// TwinCAT 3 PLC project TcTransformTest
// ProgramVersion: 3.1.4023.0
// libraries:
//   Tc2_Standard, * (Beckhoff Automation GmbH)
//   Tc2_System, * (Beckhoff Automation GmbH)
//   Tc3_Module, * (Beckhoff Automation GmbH)
//   TcMatrix, * (Burks Engineering)
//   TcTransform, * (Burks Engineering)
//   TcUnit, * (www.tcunit.org)
// project tree:
//   / PlcTask.TcTTO
//   TESTs/ FB_Vector3_Test.TcPOU, FB_RMatrix_Test.TcPOU, FB_HMatrix_Test.TcPOU, PRG_TEST.TcPOU
// real-time tasks:
//   TASK PlcTask: cycle T#10ms, priority 20, ADS port 350

CONFIGURATION TcTransformTest
    RESOURCE PLC ON TwinCAT3
        TASK PlcTask(INTERVAL := T#10ms, PRIORITY := 20);
        PROGRAM PRG_TEST WITH PlcTask : PRG_TEST;
    END_RESOURCE
END_CONFIGURATION

// ---- TESTs/PRG_TEST.TcPOU
PROGRAM PRG_TEST
VAR
	fb_Vector3 : FB_Vector3_Test;
	fb_RMatrix : FB_RMatrix_Test;
	fb_HMatrix : FB_HMatrix_Test;
END_VAR

TcUnit.RUN();

END_PROGRAM

// ---- TESTs/FB_Vector3_Test.TcPOU
FUNCTION_BLOCK FB_Vector3_Test EXTENDS FB_TestSuite
VAR_INPUT
END_VAR
VAR_OUTPUT
END_VAR
VAR
END_VAR

WhenSetExpectValuesRetained();
WhenReversedExpectValuesReversed();
WhenCrossedExpectVectorOrthogonal();
WhenParallelCrossedExpectCleared();
WhenDottedExpectResult();

METHOD PRIVATE WhenCrossedExpectVectorOrthogonal
VAR_INPUT
END_VAR
VAR
	V1 : Vector3;
	V2 : Vector3;
	V3 : Vector3;
END_VAR
TEST('WhenCrossedExpectVectorOrthogonal');

// @TEST-RUN
V1.SetFromComponents(1,0,0);
V2.SetFromComponents(0,1,0);
V3 := V1.GetVector3CrossProduct(V2);

// @TEST-ASSERT
AssertTrue(V3.Z = 1,'cross product did not work');

TEST_FINISHED();
END_METHOD

METHOD PRIVATE WhenDottedExpectResult
VAR_INPUT
END_VAR
VAR
	V1 : Vector3;
	V2 : Vector3;
	V3 : Vector3;
	Dot : LREAL;
END_VAR
TEST('WhenDottedExpectResult');

// @TEST-RUN
V1.SetFromComponents(1,2,3);
V2 := V1;
Dot := V1.GetVector3DotProduct(V2);

// @TEST-ASSERT
AssertTrue(Dot = 14,'dot product did not work');

TEST_FINISHED();
END_METHOD

METHOD PRIVATE WhenParallelCrossedExpectCleared
VAR_INPUT
END_VAR
VAR
	V1 : Vector3;
	V2 : Vector3;
	V3 : Vector3;
END_VAR
TEST('WhenParallelCrossedExpectCleared');

// @TEST-RUN
V1.SetFromComponents(1,0,0);
V2.SetFromComponents(1,0,0);
V3 := V1.GetVector3CrossProduct(V2);

// @TEST-ASSERT
AssertTrue(V3.IsCleared,'parallel cross product is not zero');

TEST_FINISHED();
END_METHOD

METHOD PRIVATE WhenReversedExpectValuesReversed
VAR_INPUT
END_VAR
VAR
	V1 : Vector3;
	V2 : Vector3;
	V3 : Vector3;
END_VAR
TEST('WhenReversedExpectValuesReversed');

// @TEST-RUN
V1.SetFromComponents(1,2,3);
V2 := V1;
V1 := V1.GetReversed();//tests getter and reverse function
V3 := V2.GetVector3Sum(V2);

// @TEST-ASSERT
AssertTrue(V2.X + V1.X = 0,'Reversal did not work');
AssertTrue(V3.X = 2,'vector sum did not work');

TEST_FINISHED();
END_METHOD

METHOD PRIVATE WhenSetExpectValuesRetained
VAR_INPUT
END_VAR
VAR
	V1 : Vector3;
	V2 : Vector3;
	V3 : DynamicMatrix;
END_VAR
TEST('WhenSetExpectValuesRetained');

// @TEST-RUN
V1.SetFromComponents(1,2,3);
V2 := V1;
V1.Clear();
V3.InitVector(3,1,1);

// @TEST-ASSERT
AssertTrue(V2.z = 3,'Component access not retained');
AssertTrue(V2.IsEqual(V3),'vector did not copy');

TEST_FINISHED();
END_METHOD

END_FUNCTION_BLOCK

// ---- TESTs/FB_RMatrix_Test.TcPOU
FUNCTION_BLOCK FB_RMatrix_Test EXTENDS FB_TestSuite
VAR_INPUT
END_VAR
VAR_OUTPUT
END_VAR
VAR
END_VAR

WhenSetFromAngleExpectResult();
WhenRotatedByIdentityExpectSame();
WhenRotatedTwiceExpectDouble();
WhenSetFrom321AnglesExpectResult();
WhenVectorRotatedExpectResult();
WhenReversedExpectOpposite();
WhenSetFromVectorsExpectResult();
WhenPostMultipliedByRMatrixExpectResult();
WhenPostMultipliedByVector3ExpectResult();

METHOD PRIVATE WhenPostMultipliedByRMatrixExpectResult
VAR_INPUT
END_VAR
VAR
	R1 : RMatrix;
	R2 : RMatrix;
R3 : RMatrix;

    Delta : LREAL := 1E-09;
END_VAR
TEST('WhenPostMultipliedByRMatrixExpectResult');

// @TEST-RUN
R1.SetFromAngle(-PI/2,0);
R1.SetFromAngle( PI/2,1);
R1.SetFromAngle(-PI/4,2);
R2.SetFromAngle( PI/3,0);

RMatrix_Product(R1, R2, R3);

// @TEST-ASSERT
AssertEquals_LREAL(0.7071067811865476, R3.GetI(0), Delta, 'R1*R2 is not correct');
AssertEquals_LREAL(0.35355339059327382071, R3.GetI(1), Delta, 'R1*R2 is not correct');
AssertEquals_LREAL(-0.61237243569579447035, R3.GetI(2), Delta, 'R1*R2 is not correct');
AssertEquals_LREAL(-0.7071067811865475, R3.GetI(3), Delta, 'R1*R2 is not correct');
AssertEquals_LREAL(0.35355339059327387071, R3.GetI(4), Delta, 'R1*R2 is not correct');
AssertEquals_LREAL(-0.61237243569579455695, R3.GetI(5), Delta, 'R1*R2 is not correct');
AssertEquals_LREAL(0, R3.GetI(6), Delta, 'R1*R2 is not correct');
AssertEquals_LREAL(0.8660254037844386, R3.GetI(7), Delta, 'R1*R2 is not correct');
AssertEquals_LREAL(0.5000000000000001, R3.GetI(8), Delta, 'R1*R2 is not correct');

TEST_FINISHED();
END_METHOD

METHOD PRIVATE WhenPostMultipliedByVector3ExpectResult
VAR_INPUT
END_VAR
VAR
	R1 : RMatrix;
	V1 : Vector3;
    VRes : Vector3;

    Delta : LREAL := 1E-09;
END_VAR
TEST('WhenPostMultipliedByVector3ExpectResult');

// @TEST-RUN
R1.SetFromAngle(-PI/2,0);
R1.SetFromAngle( PI/2,1);
R1.SetFromAngle(-PI/4,2);

V1.SetI(0, -3);
V1.SetI(1, 7.5);
V1.SetI(2, -0.6);

RMatrix_Vector3_Product(R1, V1, VRes);

// @TEST-ASSERT
AssertEquals_LREAL(3.18198051533946345, VRes.GetI(0), Delta, 'R1*V1 is not correct');
AssertEquals_LREAL(7.4246212024587495, VRes.GetI(1), Delta, 'R1*V1 is not correct');
AssertEquals_LREAL(-0.6, VRes.GetI(2), Delta, 'R1*V1 is not correct');

TEST_FINISHED();
END_METHOD

METHOD PRIVATE WhenReversedExpectOpposite
VAR_INPUT
END_VAR
VAR
	R1 : RMatrix;
	R2 : RMatrix;
END_VAR
TEST('WhenReversedExpectOpposite');

// @TEST-RUN
R1.SetFromAngle(-PI/2,0);
R2.SetFromAngle(PI/2,0);
R2.Reverse();

// @TEST-ASSERT
AssertTrue(R2.IsEqual(R1),'Reversed R is not correct');

TEST_FINISHED();
END_METHOD

METHOD PRIVATE WhenRotatedByIdentityExpectSame
VAR_INPUT
END_VAR
VAR
	R1 : RMatrix;
	R2 : RMatrix;
END_VAR
TEST('WhenRotatedByIdentityExpectSame');

// @TEST-RUN
R1.RotateBy(R2);

// @TEST-ASSERT
AssertTrue(R1.IsEqual(R2),'Result is not the same');
AssertTrue(R2.GetDeterminant() = 1,'Determinant is not 1');

TEST_FINISHED();
END_METHOD

METHOD PRIVATE WhenRotatedTwiceExpectDouble
VAR_INPUT
END_VAR
VAR
	R1 : RMatrix;
	R2 : RMatrix;
	R3 : RMatrix;
END_VAR
TEST('WhenRotatedTwiceExpectDouble');

// @TEST-RUN
R1.SetFromAngle(PI/2,0);
R2.RotateBy(R1);
R2.RotateBy(R1);
R1.SetFromAngle(PI,0);
R3.RotateBy(R1);

// @TEST-ASSERT
AssertTrue(R3.IsEqual(R2),'Results are not identical');
AssertTrue(R2.GetRC(1,1) = -1,'Y Axis not reversed');
AssertTrue(R2.GetRC(2,2) = -1,'Z Axis not reversed');

TEST_FINISHED();
END_METHOD

METHOD PRIVATE WhenSetFrom321AnglesExpectResult
VAR_INPUT
END_VAR
VAR
	A1 : TaitBryanAngleOrientation;
	A2 : TaitBryanAngleOrientation;
	R1 : RMatrix;
	R2 : RMatrix;
	R3 : RMatrix;
END_VAR
TEST('WhenSetFrom321AnglesExpectResult');

// @TEST-RUN
A1.SetFromComponentsRad(PI/2,PI/2,PI/2,TaitBryanAngleSequence.ZYX);
R1 := A1.GetRMatrix();
R2.SetFromAngle(PI/2,0);
R3.RotateBy(R2);
R2.SetFromAngle(PI/2,1);
R3.RotateBy(R2);
R2.SetFromAngle(PI/2,2);
R3.RotateBy(R2);
A2 := R1.GetAngleSequence();

// @TEST-ASSERT
AssertTrue(R1.IsEqual(R3),'rotations from two methods are not equal');
AssertTrue(R1.GetRC(0,2) = 1,'R1 X vector not correct');
AssertTrue(R1.GetRC(1,1) = 1,'R1 Y vector not correct');
AssertTrue(R1.GetRC(2,0) = -1,'R1 Z vector not correct');
AssertTrue(R1.GetDeterminant() = 1,'R1 Determinant is not 1');

AssertTrue(R3.GetRC(0,2) = 1,'R3 X vector not correct');
AssertTrue(R3.GetRC(1,1) = 1,'R3 Y vector not correct');
AssertTrue(R3.GetRC(2,0) = -1,'R3 Z vector not correct');
AssertTrue(R3.GetDeterminant() = 1,'R3 Determinant is not 1');

TEST_FINISHED();
END_METHOD

METHOD PRIVATE WhenSetFromAngleExpectResult
VAR_INPUT
END_VAR
VAR
	R1 : RMatrix;
	R2 : RMatrix;
	R3 : RMatrix;
	R4 : RMatrix;
END_VAR
TEST('WhenSetFromAngleExpectResult');

// @TEST-RUN
R1.SetFromAngle(PI/2,0);
R2.SetFromAngle(PI/2,1);
R3.SetFromAngle(PI/2,2);
R4 := R3;
R3.Clear();

// @TEST-ASSERT
AssertTrue(R1.GetRC(0,0) = 1,'R1 X vector not correct');
AssertTrue(R1.GetRC(1,2) = -1,'R1 Y vector not correct');
AssertTrue(R1.GetRC(2,1) = 1,'R1 Z vector not correct');
AssertTrue(R1.GetDeterminant() = 1,'R1 Determinant is not 1');

AssertTrue(R2.GetRC(0,2) = 1,'R2 X vector not correct');
AssertTrue(R2.GetRC(1,1) = 1,'R2 Y vector not correct');
AssertTrue(R2.GetRC(2,0) = -1,'R2 Z vector not correct');
AssertTrue(R2.GetDeterminant() = 1,'R2 Determinant is not 1');

AssertTrue(R4.GetRC(0,1) = -1,'R4 X vector not correct');
AssertTrue(R4.GetRC(1,0) = 1,'R4 Y vector not correct');
AssertTrue(R4.GetRC(2,2) = 1,'R4 Z vector not correct');
AssertTrue(R4.GetDeterminant() = 1,'R4 Determinant is not 1');

TEST_FINISHED();
END_METHOD

METHOD PRIVATE WhenSetFromVectorsExpectResult
VAR_INPUT
END_VAR
VAR
	VX : Vector3;
	VY : Vector3;
	VZ : Vector3;
	R1 : RMatrix;
	RX : RMatrix;
	RY : RMatrix;
	RZ : RMatrix;
	RBad : RMatrix;
	
	ResX : BOOL;
	ResY : BOOL;
	ResZ : BOOL;
	ResBad : BOOL;
END_VAR
TEST('WhenSetFromVectorsExpectResult');

// @TEST-RUN
R1.SetFromAngle(PI/2,1);//90 deg rotation around Y
VX.SetFromComponents(0,0,-1);
VY.SetFromComponents(0,1,0);
VZ.SetFromComponents(1,0,0);
RX.SetFromVectorsYZ(VY,VZ);
RY.SetFromVectorsXZ(VX,VZ);
RZ.SetFromVectorsXY(VX,VY);
Rbad.SetFromVectorsXY(VX,VX);

// @TEST-ASSERT
AssertTrue(R1.IsNearlyEqual(RX,1E-9),'RX not calculated correctly');
AssertTrue(R1.IsNearlyEqual(RY,1E-9),'RY not calculated correctly');
AssertTrue(R1.IsNearlyEqual(RZ,1E-9),'RZ not calculated correctly');

TEST_FINISHED();
END_METHOD

METHOD PRIVATE WhenVectorRotatedExpectResult
VAR_INPUT
END_VAR
VAR
	R1 : RMatrix;
	V1 : Vector3;
	V2 : Vector3;
END_VAR
TEST('WhenVectorRotatedExpectResult');

// @TEST-RUN
R1.SetFromAngle(PI/2,1);
V1.X := 1;
V2 := R1.GetRotatedVector3(V1);

// @TEST-ASSERT
AssertTrue(V2.Z = -1,'Result is not in correct direction');
AssertTrue(V2.GetVectorMagnitude() = 1,'magnitude is not 1');

TEST_FINISHED();
END_METHOD

END_FUNCTION_BLOCK

// ---- TESTs/FB_HMatrix_Test.TcPOU
FUNCTION_BLOCK FB_HMatrix_Test EXTENDS FB_TestSuite
VAR_INPUT
END_VAR
VAR_OUTPUT
END_VAR
VAR
END_VAR

WhenSetFromComponentsExpectValuesRetained();
WhenTransformedByIdentityExpectSame();
WhenVectorTransformedExpectResult();
WhenMatrixTransformedExpectResult();
WhenPostMultipliedByHMatrixExpectResult();

METHOD PRIVATE WhenMatrixTransformedExpectResult
VAR_INPUT
END_VAR
VAR
	H1 : HMatrix;
	H2 : HMatrix;
	H3 : HMatrix;
	R1 : RMatrix;
	V1 : Vector3;
	V2 : Vector3;
	V3 : Vector3;
	V4 : Vector3;
END_VAR
TEST('WhenMatrixTransformedExpectResult');

// @TEST-RUN
R1.SetFromAngle(PI/2,1);
V1.X := 1;
H1.SetFromComponents(R1,V1);
H2 := H1;
H3 := H1.GetTransformedHMatrix(H2);

V2.SetFromComponents(1,0,0);
V3 := H3.GetTransformedVector3(V2);
V4.SetFromComponents(0,0,-1);

// @TEST-ASSERT
AssertTrue(V3.IsNearlyEqual(V4,1E-6),'Result is not correct');

TEST_FINISHED();
END_METHOD

METHOD WhenPostMultipliedByHMatrixExpectResult
VAR_INPUT
END_VAR
VAR
	H1 : HMatrix;
	H2 : HMatrix;
    H3 : HMatrix;

    R1 : RMatrix;
    R2 : RMatrix;

    V1 : Vector3;
    V2 : Vector3;

    Delta : LREAL := 1E-09;
END_VAR
TEST('WhenPostMultipliedByHMatrixExpectResult');

// @TEST-RUN
R1.SetFromAngle(-PI/3,0);
R1.SetFromAngle( PI/5,1);
R1.SetFromAngle(-PI/6,2);
V1.SetI(0, -3);
V1.SetI(1, 7.5);
V1.SetI(2, -0.6);

R2.SetFromAngle(PI/7,0);
R2.SetFromAngle(-PI/3,1);
R2.SetFromAngle(PI/5,2);
V2.SetI(0, 15.1);
V2.SetI(1, -0.34);
V2.SetI(2, 5.75);

H1.SetFromComponents(R1, V1);
H2.SetFromComponents(R2, V2);

HMatrix_Product(H1, H2, H3);

// @TEST-ASSERT
AssertEquals_LREAL(0.99452189536827339586,  H3.GetI(0), Delta, 'H1*H2 is not correct');
AssertEquals_LREAL(-0.10452846326765348803, H3.GetI(1), Delta, 'H1*H2 is not correct');
AssertEquals_LREAL(0,                       H3.GetI(2), Delta, 'H1*H2 is not correct');
AssertEquals_LREAL(9.90698359714502437,     H3.GetI(3), Delta, 'H1*H2 is not correct');
AssertEquals_LREAL(0.10452846326765348803,  H3.GetI(4), Delta, 'H1*H2 is not correct');
AssertEquals_LREAL(0.99452189536827339586,  H3.GetI(5), Delta, 'H1*H2 is not correct');
AssertEquals_LREAL(0,                       H3.GetI(6), Delta, 'H1*H2 is not correct');
AssertEquals_LREAL(-0.344448637286709158,   H3.GetI(7), Delta, 'H1*H2 is not correct');
AssertEquals_LREAL(0,                       H3.GetI(8), Delta, 'H1*H2 is not correct');
AssertEquals_LREAL(0,                       H3.GetI(9), Delta, 'H1*H2 is not correct');
AssertEquals_LREAL(1,                       H3.GetI(10), Delta, 'H1*H2 is not correct');
AssertEquals_LREAL(5.15,                    H3.GetI(11), Delta, 'H1*H2 is not correct');
AssertEquals_LREAL(0,                       H3.GetI(12), Delta, 'H1*H2 is not correct');
AssertEquals_LREAL(0,                       H3.GetI(13), Delta, 'H1*H2 is not correct');
AssertEquals_LREAL(0,                       H3.GetI(14), Delta, 'H1*H2 is not correct');
AssertEquals_LREAL(1,                       H3.GetI(15), Delta, 'H1*H2 is not correct');

TEST_FINISHED();
END_METHOD

METHOD PRIVATE WhenSetFromComponentsExpectValuesRetained
VAR_INPUT
END_VAR
VAR
	R1 : RMatrix;
	R2 : RMatrix;
	V1 : Vector3;
	V2 : Vector3;
	H1 : HMatrix;
	H2 : HMatrix;
END_VAR
TEST('WhenSetFromComponentsExpectValuesRetained');

// @TEST-RUN
R1.SetFromAngle(PI/2,0);
V1.SetFromComponents(1,2,3);
H1.SetFromComponents(R1,V1);
H2 := H1;
H1.Clear();
R2 := H2.RMatrixComponent;
V2 := H2.Vector3Component;
// @TEST-ASSERT
AssertTrue(R1.IsEqual(R2),'Rotation component not correct');
AssertTrue(V1.IsEqual(V2),'Vector component not correct');

TEST_FINISHED();
END_METHOD

METHOD PRIVATE WhenTransformedByIdentityExpectSame
VAR_INPUT
END_VAR
VAR
	H1 : HMatrix;
	H2 : HMatrix;
	H3 : HMatrix;
	R1 : RMatrix;
	V1 : Vector3;
END_VAR
TEST('WhenTransformedByIdentityExpectSame');

// @TEST-RUN
R1.SetFromAngle(PI/2,0);
V1.SetFromComponents(1,2,3);
H1.SetFromComponents(R1,V1);
H3 := H1;
H1.TransformBy(H2);

// @TEST-ASSERT
AssertTrue(H1.IsEqual(H3),'Result is not the same');

TEST_FINISHED();
END_METHOD

METHOD PRIVATE WhenVectorTransformedExpectResult
VAR_INPUT
END_VAR
VAR
	H1 : HMatrix;
	R1 : RMatrix;
	V1 : Vector3;
	V2 : Vector3;
	V3 : Vector3;
	V4 : Vector3;
END_VAR
TEST('WhenVectorTransformedExpectResult');

// @TEST-RUN
R1.SetFromAngle(PI/2,1);//90deg rotation around Y axis
V1.X := 1;
H1.SetFromComponents(R1,V1);
V2.X := 1;
V3 := H1.GetTransformedVector3(V2);
V4.SetFromComponents(1,0,-1);

// @TEST-ASSERT
AssertTrue(V3.IsEqual(V4),'Result is not correct');

TEST_FINISHED();
END_METHOD

END_FUNCTION_BLOCK
